// TIA Portal project "TIA-Prgm-ATV630-rv3" (V15.1)

(* hardware
DEVICE "S7-1200 station_1"  S7-1200 Station
   slot 0: "Rack_0"  S7-1200 Rack  Rack  V1.0
   slot 1: "PLC_1"  CPU 1215C DC/DC/DC  6ES7 215-1AG40-0XB0  V4.0
DEVICE "GSD device_2"  GSD.Device.PN
   slot 0: "Rack"  Rack  V1.0
   slot 0: "ATV630"  ATV630  ATV630
      slot 0: "ATV630"  ATV630
      slot 1: "Interface"  Interface
         slot 1: "Port 1"  Port 1
         slot 2: "Port 2"  Port 2
   slot 1: "Telegram 101 (4PKW/6PZD)_1"  Telegram 101 (4PKW/6PZD)
      slot 0: "Telegram 101"  Telegram 101
*)

// ===== PLC "PLC_1"  CPU 1215C DC/DC/DC =====
// protected blocks, not shown: "ATV630_rv3"

VAR_GLOBAL   // PLC tag table "VFD_Tags"
   "Status_Word" AT %IW76 : Word;   // Drive Status Word
   "Motor_Rpms_In" AT %IW78 : Int;   // Here if you need it. Not in this block
   "Amps_In" AT %IW82 : UInt;   // Amps feedback from drive
   "Fault_Code" AT %IW84 : Word;   // Fault code from drive
   "Control_Word" AT %QW76 : Word;   // Control word to drive
   "Speed_Out_Hz" AT %QW78 : Int;   // Output Speed setpoint to Drive.
   "Run_Fwd" AT %M0.0 : Bool;
   "Run_Rev" AT %M0.1 : Bool;
   "Reset_Fault" AT %M0.2 : Bool;
   "Enable" AT %M0.3 : Bool;
   "Amps_Out" AT %MD0 : Real;
   "Stop" AT %M0.4 : Bool;
   "Line_Volts_In" AT %IW80 : UInt;   // Line voltage reading from drive
   "Speed_Setpoint_Hz" AT %MD4 : Real;   // Set desired speed in Hz `00.0Hz to 60.0Hz`
   "Freq_Fdbk_In" AT %IW86 : Word;   // Frequency feedback from drive
   "E_Stop" AT %M8.0 : Bool;
END_VAR

ORGANIZATION_BLOCK "Main"   // OB1, LAD, ProgramCycle
TITLE = "Main Program Sweep (Cycle)"
{ S7_Optimized_Access := 'TRUE' }
VERSION : 0.1
   VAR_INPUT
      Initial_Call : Bool;   // Initial call of this OB
      Remanence : Bool;   // =True, if remanent data are available
   END_VAR
BEGIN

REGION Network 1
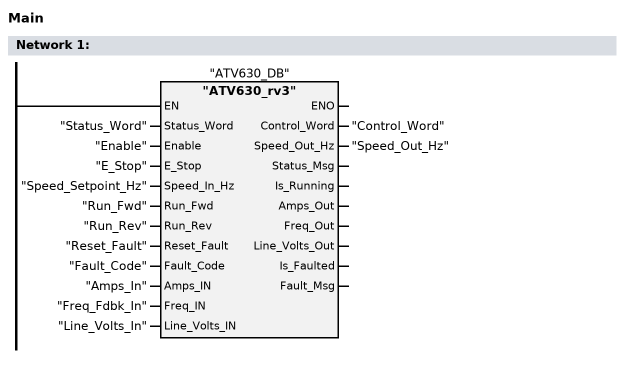
   RUNG wire#powerrail
      "ATV630_DB"(Status_Word := "Status_Word", Enable := "Enable", E_Stop := "E_Stop", Speed_In_Hz := "Speed_Setpoint_Hz", Run_Fwd := "Run_Fwd", Run_Rev := "Run_Rev", Reset_Fault := "Reset_Fault", Fault_Code := "Fault_Code", Amps_IN := "Amps_In", Freq_IN := "Freq_Fdbk_In", Line_Volts_IN := "Line_Volts_In", Control_Word => "Control_Word", Speed_Out_Hz => "Speed_Out_Hz", Status_Msg =>, Is_Running =>, Amps_Out =>, Freq_Out =>, Line_Volts_Out =>, Is_Faulted =>, Fault_Msg =>)
   END_RUNG
   // the same network as SCL:
   "ATV630_DB"(Status_Word := "Status_Word",   // "ATV630_rv3"
               Enable := "Enable",
               E_Stop := "E_Stop",
               Speed_In_Hz := "Speed_Setpoint_Hz",
               Run_Fwd := "Run_Fwd",
               Run_Rev := "Run_Rev",
               Reset_Fault := "Reset_Fault",
               Fault_Code := "Fault_Code",
               Amps_IN := "Amps_In",
               Freq_IN := "Freq_Fdbk_In",
               Line_Volts_IN := "Line_Volts_In",
               Control_Word => "Control_Word",
               Speed_Out_Hz => "Speed_Out_Hz");
END_REGION
END_ORGANIZATION_BLOCK